KUKA KRL program: ABA_MESA_B.src

&ACCESS RV
&PARAM EDITMASK = *
&PARAM TEMPLATE = C:\KRC\Roboter\Template\FunctionVorgabe
DEFFCT BOOL ABA_MESA_B( )

ENDFCT
